(* CODESYS project temp.project

Project tree, tasks and I/O mapping:
  Device : XV100, Eaton Automation, version 3.5.4.0
    application PLC_Main
      libraries: Standard, * (System); IoDrvModbusSerialSlave, 3.5.3.80 (3S - Smart Software Solutions GmbH); Util, 3.5.1.0 (System); EA_CANopen, 3.5.2.0 (Eaton Automation); CAA File, 3.5.3.0 (CAA Technical Workgroup)
      task MainTask (cyclic, interval t#10ms, priority 1) calls PLC_PRG
      program PLC_PRG [ST]
      global variables GVL
      Symbols
      trace Trace (task MainTask, trigger Positive on PLC_PRG.blinkOut): param::Device.Modbus_COM.Modbus_Master_COM_Port.IOModule:1:2100000.Trigger:Channel 1.Trigger, param::Device.Modbus_COM.Modbus_Master_COM_Port.ROBKO_01:1:2100000.Trigger:Channel 2.Trigger
      function ROBKO01_JOG [ST]
      function File_Standard_EXAMPLE [ST]
      function Robko01_Forward_Kinematics_From_Motor_Pos [ST]
      global variables ROBKO
      function degrees [ST]
    Modbus_COM : Modbus COM, 3S - Smart Software Solutions GmbH, version 3.4.0.0
        settings: DataBits = 8; StopBits = 2; ComPort = 1
      Modbus_Master_COM_Port : Modbus Master, COM Port, 3S - Smart Software Solutions GmbH, version 3.5.4.0
          settings: Transmission = 'RTU'; ResponseTimeout = 500; TimeBetweenFrames = 20
        IOModule : Modbus Slave, COM Port, 3S - Smart Software Solutions GmbH, version 3.5.4.0
            settings: SlaveAddress = 10; ResponseTimeout = 500; UseExtendedFunctionCodes = TRUE; Channel 2.Function Code = 15; Channel 2.Read Offset = 0; Channel 2.Read Length = 0; Channel 2.Write Offset = 16#0000; Channel 2.Write Length = 12; Channel 2.Cycle Time = 100; Channel 1.Function Code = 2; Channel 1.Read Offset = 16#0000; Channel 1.Read Length = 11; Channel 1.Write Offset = 0; Channel 1.Write Length = 0; Channel 1.Cycle Time = 100
            output IOModule_Q0 : BOOL  // Channel 2.Channel 2[0].Bit0
            output IOModule_Q1 : BOOL  // Channel 2.Channel 2[0].Bit1
            output IOModule_Q2 : BOOL  // Channel 2.Channel 2[0].Bit2
            output IOModule_Q3 : BOOL  // Channel 2.Channel 2[0].Bit3
            output IOModule_Q4 : BOOL  // Channel 2.Channel 2[0].Bit4
            output IOModule_Q5 : BOOL  // Channel 2.Channel 2[0].Bit5
            output IOModule_Q6 : BOOL  // Channel 2.Channel 2[0].Bit6
            output IOModule_Q7 : BOOL  // Channel 2.Channel 2[0].Bit7
            output IOModule_Q8 : BOOL  // Channel 2.Channel 2[1].Bit0
            output IOModule_Q9 : BOOL  // Channel 2.Channel 2[1].Bit1
            output IOModule_Q10 : BOOL  // Channel 2.Channel 2[1].Bit2
            output IOModule_Q11 : BOOL  // Channel 2.Channel 2[1].Bit3
            input  IOModule_I0 : BOOL  // Channel 1.Channel 1[0].Bit0
            input  IOModule_I1 : BOOL  // Channel 1.Channel 1[0].Bit1
            input  IOModule_I2 : BOOL  // Channel 1.Channel 1[0].Bit2
            input  IOModule_I3 : BOOL  // Channel 1.Channel 1[0].Bit3
            input  IOModule_I4 : BOOL  // Channel 1.Channel 1[0].Bit4
            input  IOModule_I5 : BOOL  // Channel 1.Channel 1[0].Bit5
            input  IOModule_I6 : BOOL  // Channel 1.Channel 1[0].Bit6
            input  IOModule_I7 : BOOL  // Channel 1.Channel 1[0].Bit7
            input  IOModule_I8 : BOOL  // Channel 1.Channel 1[1].Bit0
            input  IOModule_I9 : BOOL  // Channel 1.Channel 1[1].Bit1
            input  IOModule_I10 : BOOL  // Channel 1.Channel 1[1].Bit2
            unmapped channels: Channel 2, Channel 1
        ROBKO_01 : Modbus Slave, COM Port, 3S - Smart Software Solutions GmbH, version 3.5.4.0
            settings: SlaveAddress = 11; ResponseTimeout = 50; UseExtendedFunctionCodes = TRUE; Channel 1.Function Code = 4; Channel 1.Read Offset = 16#0000; Channel 1.Read Length = 13; Channel 1.Write Offset = 0; Channel 1.Write Length = 0; Channel 1.Cycle Time = 95; Channel 2.Function Code = 15; Channel 2.Read Offset = 0; Channel 2.Read Length = 0; Channel 2.Write Offset = 16#0000; Channel 2.Write Length = 12; Channel 2.Cycle Time = 100; ROBKO_WRITE_CONTROL_REGISTER_6.Function Code = 6; ROBKO_WRITE_CONTROL_REGISTER_6.Read Offset = 0; ROBKO_WRITE_CONTROL_REGISTER_6.Read Length = 0; ROBKO_WRITE_CONTROL_REGISTER_6.Write Offset = 16#0006; ROBKO_WRITE_CONTROL_REGISTER_6.Write Length = 1; ROBKO_WRITE_CONTROL_REGISTER_6.Cycle Time = 100; Channel 3.Function Code = 16; Channel 3.Read Offset = 0; Channel 3.Read Length = 0; Channel 3.Write Offset = 16#0000; Channel 3.Write Length = 13; Channel 3.Cycle Time = 100
            input  t : ARRAY[0..12] OF WORD  // Channel 1
            output JOG1_DIRECTION : BOOL  // Channel 2.Channel 2[0].Bit0
            output JOG2_DIRECTION : BOOL  // Channel 2.Channel 2[0].Bit1
            output JOG3_DIRECTION : BOOL  // Channel 2.Channel 2[0].Bit2
            output JOG4_DIRECTION : BOOL  // Channel 2.Channel 2[0].Bit3
            output JOG5_DIRECTION : BOOL  // Channel 2.Channel 2[0].Bit4
            output JOG6_DIRECTION : BOOL  // Channel 2.Channel 2[0].Bit5
            output JOG1 : BOOL  // Channel 2.Channel 2[0].Bit6
            output JOG2 : BOOL  // Channel 2.Channel 2[0].Bit7
            output JOG3 : BOOL  // Channel 2.Channel 2[1].Bit0
            output JOG4 : BOOL  // Channel 2.Channel 2[1].Bit1
            output JOG5 : BOOL  // Channel 2.Channel 2[1].Bit2
            output JOG6 : BOOL  // Channel 2.Channel 2[1].Bit3
            output ROBKO_WRITE_CONTROL_REGISTER_TRIGER AT %QX4.0 : BIT  // ROBKO_WRITE_CONTROL_REGISTER_6
            output ROBKO_CONTROL_REGISTER : WORD  // ROBKO_WRITE_CONTROL_REGISTER_6.ROBKO_WRITE_CONTROL_REGISTER_6[0]
            output ROBKO : ARRAY[0..12] OF WORD  // Channel 3
            unmapped channels: Channel 2, ROBKO_WRITE_CONTROL_REGISTER_6, %QX8.0 Channel 3
*)

// Device/PLC_Main/GVL
VAR_GLOBAL
	HMI_Byte_1					: BYTE;
	HMI_Button_1				: BYTE;
	
	HMI_blinkEnable				: BYTE  :=  0;	
	HMI_Blink_Time_Low			: WORD  :=  100;
	HMI_Blink_Time_High			: WORD  :=  100;
	
	HMI_ROBKO_Button_SetZeroPos	: BYTE  :=  0;
	HMI_ROBKO_JogByte			: BYTE  :=  0;
	HMI_ROBKO_JOG_Switch		: BYTE  :=  1;
	HMI_ROBKO_JOG_Pos			: BYTE  :=  0;
	HMI_ROBKO_JOG_Neg			: BYTE  :=  0;
	
	HMI_ROBKO_G01_X				: INT  :=  0;
	HMI_ROBKO_G01_Y				: INT  :=  0;
	HMI_ROBKO_G01_Z				: INT  :=  0;
	HMI_ROBKO_G01_BUTTON		: BYTE;

	HMI_ROBKO_ARR_POS			: ARRAY [ 0..5 ] OF REAL;
	
	test11 : BOOL;
	
	
	
	
	
	xFileStdInit:			BOOL := FALSE;
	uiFileStdState:			UINT := 0;
	sFileName:				FILE.CAA.FILENAME := '\Test.txt';
	hFile:					FILE.CAA.HANDLE;

	sFileTestString:		STRING := 'Hello caa library user';

	sFileString:			STRING := '';
	szFileSize1:			FILE.CAA.SIZE  :=  0;
	szFileSize2:			FILE.CAA.SIZE  :=  0;

	file_get_root:			FILE.GetRoot;
	filop:					FILE.Open;
	filwr:					FILE.Write;
	filrd:					FILE.Read;
	filcl:					FILE.Close;
END_VAR

// Device/PLC_Main/ROBKO
VAR_GLOBAL
// Motor Consts [ Steps / Rad ]:
	T1const		: REAL := 1222.7;
	T2const		: REAL := 1145.915; //1161.4f;
	T3const		: REAL := 668.4507; //680.1f
	T4const		: REAL := 244.7;
	T5const		: REAL := 244.7;
	T6const		: REAL := 2.0 * 270.0;

	H			: REAL := 195.0;
	L1			: REAL := 178.0;
	L2			: REAL := 178.0;
	LG			: REAL := 92.0;

	R1			: REAL := 0.0;
	C			: REAL := 180.0 / 3.14;
END_VAR

// Device/PLC_Main/PLC_PRG
PROGRAM PLC_PRG
VAR
	i			: INT  :=  1;	
	temp		: INT;
	flag		: BYTE;
	
	flash		: BLINK;
	blinkOut	: BOOL;
	
	TR_ON_BUTTON_1	: R_TRIG;

	TR_ON_BUTTON_ROBKO_01_G01	: R_TRIG;
	
	R_TRIG_IOModuleResetError : R_TRIG;
	R_TRIG_ROBKO_ResetError : R_TRIG;
	
	R_TRIG_Button_SetZeroPos : R_TRIG;
	R_TRIG_ROBKO_WRITE_CONTROL_REGISTER : R_TRIG;
	
	temp1 : ARRAY[ 0..12 ] OF INT;
	
	arrMotor : ARRAY[ 0..5 ] OF INT;
	
	j : INT;
	
	x : BYTE;
	
	uiTemp : UINT;
	
END_VAR

R_TRIG_IOModuleResetError( clk  :=  IOModule.xError, Q=> IOModule.xReset );
R_TRIG_ROBKO_ResetError( clk  :=  ROBKO_01.xError, Q=> ROBKO_01.xReset );

//File_Standard_EXAMPLE();

TR_ON_BUTTON_1( clk  :=  BYTE_TO_BOOL(HMI_Button_1), Q => );

IF TR_ON_BUTTON_1.Q THEN
	IF HMI_blinkEnable = 0 THEN
		HMI_blinkEnable  :=  1;
	ELSE
		HMI_blinkEnable  :=  0;
	END_IF
END_IF

i  :=  i + 1;
HMI_Byte_1  :=  INT_TO_BYTE( i );

IF i > 100 THEN
	i  :=  0;

	IF flag = 0 THEN
		flag  :=  1;
	ELSE
		flag  :=  0;
	END_IF

END_IF

IF flag = 0 THEN
	IOModule_Q0  :=  FALSE;
	IOModule_Q9  :=  TRUE;
ELSE
	IOModule_Q0  :=  TRUE;
	IOModule_Q9  :=  FALSE;
END_IF

IF HMI_blinkEnable = 1 THEN
	IOModule_Q3  :=  blinkOut;
ELSE
	IOModule_Q3  :=  FALSE;
END_IF

flash
(
	ENABLE		 :=  TRUE,
	TIMELOW		 :=  WORD_TO_TIME( HMI_Blink_Time_Low ),
	TIMEHIGH	 :=  WORD_TO_TIME( HMI_Blink_Time_High ),
	OUT			=> blinkOut
);

(* ------------------------------------------------------------------------------------------------------------------------------------- *)

TR_ON_BUTTON_ROBKO_01_G01( clk  :=  BYTE_TO_BOOL( HMI_ROBKO_G01_BUTTON ), Q=> );

IF TR_ON_BUTTON_ROBKO_01_G01.Q = TRUE THEN
	ROBKO[ 6 ]  :=  4 OR ( 16#0100 OR 16#0200 OR 16#0400 );
	ROBKO[ 7 ]  :=  INT_TO_WORD( HMI_ROBKO_G01_X );
	ROBKO[ 8 ]  :=  INT_TO_WORD( HMI_ROBKO_G01_Y );
	ROBKO[ 9 ]  :=  INT_TO_WORD( HMI_ROBKO_G01_Z );
END_IF

%QX8.0  :=  TR_ON_BUTTON_ROBKO_01_G01.Q;
// =================================================================================================
ROBKO01_JOG();
// =================================================================================================
R_TRIG_Button_SetZeroPos( clk  :=  BYTE_TO_BOOL( HMI_ROBKO_Button_SetZeroPos ), Q=> );

IF R_TRIG_Button_SetZeroPos.Q (* AND ROBKO_JOG_MODE *) THEN
	ROBKO_CONTROL_REGISTER  :=  3;
END_IF
// =================================================================================================
R_TRIG_ROBKO_WRITE_CONTROL_REGISTER
(
	clk  :=  R_TRIG_Button_SetZeroPos.Q,
	Q => ROBKO_WRITE_CONTROL_REGISTER_TRIGER
);
// =================================================================================================
FOR j :=  0 TO 12 BY 1 DO

	temp1[ j ]  :=  WORD_TO_INT( t[ j ] );

	IF UINT_TO_BOOL( 16#8000 AND INT_TO_UINT( temp1[ j ] ) ) THEN
		temp1[ j ]  :=  UINT_TO_INT( ( 16#7FFF AND INT_TO_UINT( temp1[ j ] ) ) - 32768 );
	END_IF

END_FOR

FOR j:= 0 TO 5 BY 1 DO
	arrMotor[ j ] := temp1[ 6 + j ];
END_FOR

Robko01_Forward_Kinematics_From_Motor_Pos( arrMotor := arrMotor, arrPos => HMI_ROBKO_ARR_POS );


// =================================================================================================

END_PROGRAM

// Device/PLC_Main/File_Standard_EXAMPLE
FUNCTION File_Standard_EXAMPLE : BOOL
VAR_INPUT
END_VAR

(*VAR
	xFileStdInit:			BOOL := FALSE;
	uiFileStdState:			UINT := 0;
	sFileName:				FILE.CAA.FILENAME := 'TestFile.txt';
	hFile:					FILE.CAA.HANDLE;

	sFileTestString:		STRING := 'Hello caa library user';

	sFileString:			STRING := '';
	szFileSize1:			FILE.CAA.SIZE  :=  0;
	szFileSize2:			FILE.CAA.SIZE  :=  0;

	filop:					FILE.Open;
	filwr:					FILE.Write;
	filrd:					FILE.Read;
	filcl:					FILE.Close;
END_VAR*)

IF NOT xFileStdInit THEN

	filop( xExecute := FALSE );
	filcl( xExecute := FALSE );
	filwr( xExecute := FALSE );
	filrd( xExecute := FALSE );

	xFileStdInit	:= TRUE;
	uiFileStdState	:= 0;

ELSE

	CASE uiFileStdState OF
	0: (* create a new file *)
		filop.sFileName := sFileName;
		filop.eFileMode := FILE.MODE.MRDWR;
		filop.xExclusive := TRUE;
		filop( xExecute := TRUE);
		
		WHILE filop.xDone = FALSE DO
			;
		END_WHILE

		IF filop.xDone THEN
			hFile := filop.hFile;
			uiFileStdState := 1;
		END_IF

		IF filop.xError THEN
			(* error handling*);
		END_IF

	1: (* write text in the file *)
		filwr.hFile := hFile;
		filwr.pBuffer := ADR(sFileTestString);
		szFileSize1 := SIZEOF(sFileTestString);
		
		filwr.szSize := szFileSize1;
		filwr.udiTimeOut := 100000;	     (* 100ms Timeout *)

		filwr( xExecute := TRUE);

		IF filwr.xDone THEN
			uiFileStdState := 2;
		END_IF

		IF filwr.xError THEN
			(* error handling*);
		END_IF

	2: (* read file - TestFile.txt*)
		filrd.hFile := hFile;
		filrd.udiTimeOut := 100000;	      (* 100ms Timeout *)
		filrd.pBuffer := ADR(sFileString);
		filrd.szBuffer := 255;

		filrd( xExecute := TRUE);

		IF filrd.xDone THEN
			szFileSize2 := filrd.szSize;

			IF szFileSize2 = szFileSize1 THEN
				uiFileStdState := 3;
			ELSE
				(* error handling*);
			END_IF
		END_IF

		IF filrd.xError THEN
			(* error handling*);
		END_IF

	3: (* close file  - TestFile.txt *)
		filcl.hFile := hFile;
		filcl( xExecute := TRUE);
	
		IF filcl.xDone THEN
			uiFileStdState := 4;
		END_IF

		IF filcl.xError THEN
			(* error handling*);
		END_IF

	4: (* end of example *);
	END_CASE

END_IF

END_FUNCTION

// Device/PLC_Main/ROBKO01_JOG
FUNCTION ROBKO01_JOG : BOOL
VAR_INPUT
END_VAR
VAR
	JOGn				: BOOL;
	JOG_N_DIRECTION		: BOOL;
END_VAR

IF HMI_ROBKO_JogByte <> 0 THEN
	HMI_ROBKO_JOG_Switch  :=  HMI_ROBKO_JogByte;
	HMI_ROBKO_JogByte  :=  0; 
END_IF

IF HMI_ROBKO_JOG_Neg = 0 THEN
	JOG_N_DIRECTION  :=  FALSE;
ELSE
	JOG_N_DIRECTION  :=  TRUE;
END_IF

IF HMI_ROBKO_JOG_Pos = 1 OR HMI_ROBKO_JOG_Neg = 1 THEN
	JOGn  :=  TRUE;
ELSE
	JOGn  :=  FALSE;
END_IF

CASE HMI_ROBKO_JOG_Switch OF
	1:
		JOG1  :=  JOGn;
		JOG1_DIRECTION  :=  JOG_N_DIRECTION;

	2:
		JOG2  :=  JOGn;
		JOG2_DIRECTION  :=  JOG_N_DIRECTION;

	4:
		JOG3  :=  JOGn;
		JOG3_DIRECTION  :=  JOG_N_DIRECTION;

	8:
		JOG4  :=  JOGn;
		JOG4_DIRECTION  :=  JOG_N_DIRECTION;

	16:
		JOG5  :=  JOGn;
		JOG5_DIRECTION  :=  JOG_N_DIRECTION;

	32:
		JOG6  :=  JOGn;
		JOG6_DIRECTION  :=  JOG_N_DIRECTION;

END_CASE

END_FUNCTION

// Device/PLC_Main/Robko01_Forward_Kinematics_From_Motor_Pos
FUNCTION Robko01_Forward_Kinematics_From_Motor_Pos : BOOL
VAR_INPUT
	arrMotor	: ARRAY[0..5] OF INT;
END_VAR

VAR_OUTPUT
	arrPos		: ARRAY[0..5] OF REAL;
END_VAR
	
VAR
	XX, YY, ZZ, PP, RR, RP	: REAL;
	T1, T2, T3, T4, T5, T6	: REAL;
END_VAR

(*void Robko01_Forward_Kinematics_From_Motor_Pos
(
	int arrMotor[6],
	real arrPos[6],
	real R1
)
{
	real XX, YY, ZZ, PP, RR, RP;
	real T1 = arrMotor[0] / T1const;
	real T2 = arrMotor[1] / T2const;
	real T3 = arrMotor[2] / T3const;
	real T4 = arrMotor[3] / T4const;
	real T5 = arrMotor[4] / T5const;
	real T6 = arrMotor[5] / T6const;

	PP = ( T4 + T5 ) / 2;
	RR = ( T4 - T5 ) / 2 - R1 * T1;

	RP = L1 * (real)cos( T2 ) + L2 * (real)cos( T3 ) + LG * (real)cos( PP );
	XX = RP * (real)cos( T1 );
	YY = RP * (real)sin( T1 );
	ZZ = H - L1 * (real)sin( -T2 ) - L2 * (real)sin( -T3 ) - LG * (real)sin( -PP );

	PP = PP * C;
	RR = RR * C;

	arrPos[0] = XX;
	arrPos[1] = YY;
	arrPos[2] = ZZ;
	arrPos[3] = PP;
	arrPos[4] = -RR;
	arrPos[5] = -degrees(T6);
}*)

T1 := INT_TO_REAL( arrMotor[0] ) / T1const;
T2 := INT_TO_REAL( arrMotor[1] ) / T2const;
T3 := INT_TO_REAL( arrMotor[2] ) / T3const;
T4 := INT_TO_REAL( arrMotor[3] ) / T4const;
T5 := INT_TO_REAL( arrMotor[4] ) / T5const;
T6 := INT_TO_REAL( arrMotor[5] ) / T6const;

PP := ( T4 + T5 ) / 2.0;
RR := ( T4 - T5 ) / 2.0 - R1 * T1;

RP := L1 * COS( T2 ) + L2 * COS( T3 ) + LG * COS( PP );
XX := RP * COS( T1 );
YY := RP * SIN( T1 );
ZZ := H - L1 * SIN( -T2 ) - L2 * SIN( -T3 ) - LG * SIN( -PP );

PP := PP * C;
RR := RR * C;

arrPos[0] := XX;
arrPos[1] := YY;
arrPos[2] := ZZ;
arrPos[3] := PP;
arrPos[4] := -RR;
arrPos[5] := -degrees(T6);

END_FUNCTION

// Device/PLC_Main/degrees
FUNCTION degrees : REAL
VAR_INPUT
	rad : REAL;
END_VAR
VAR
END_VAR

degrees := rad * ( 180.0 / 3.14 );

END_FUNCTION
